{attribute 'qualified_only'}
VAR_GLOBAL CONSTANT
	TXT_FILE_MAX_STRING_LENGTH : UDINT := 300;
END_VAR

(* stored: Version 1.1.0.1, ProductVersion 3.1.4022.12
   GVL Param: Id {ec9b4ae4-4138-41d4-820d-f89bcc673a89}, ParameterList True *)
